Staubli VAL3: boolOr.pgx

public program boolOr(string x_sBinary1, string x_sBinary2, string& x_sReturn[])
  local num l_nNumBit
  local string l_sValsup
  local string l_sValmin
begin
  //-----------------------------------------------------------------------
  //Header begin
  //Description of program
  //  This program provides an Or logical operator for 2 binary values.
  //
  //     0 or 0 = 0
  //     0 or 1 = 1
  //     1 or 1 = 1
  //
  //Input parameters
  //  string x_sBinary1 :
  //    role : 1 st binary number
  //  string x_sBinary2 :
  //    role : 2 nd binary number
  //
  //Output parameters
  //  string x_sReturn :
  //    role : Result of calculation x_sBinary1 OR x_sBinary2
  //
  //Example
  //  Or("10101011","00011011",sResult)
  //
  //History
  //  Creation : 16-04-09 - t.Gra
  //Header end
  //-----------------------------------------------------------------------
  //Initialization
  l_nNumBit=0
  l_sValsup=""
  l_sValmin=""
  //call function for error control
  call ChekCompBinary(x_sBinary1,x_sBinary2,l_sValsup,l_sValmin)
  //calcul loop
  if (bRead==true)
    for l_nNumBit=(len(l_sValsup)-1) to 0 step -1
      if ((mid(l_sValsup,1,l_nNumBit)=="0") and (mid(l_sValmin,1,l_nNumBit)=="0"))
        x_sReturn="0"+x_sReturn
      else
        x_sReturn="1"+x_sReturn
      endIf
    endFor
  else
    x_sReturn="Error"
  endIf
end
